FUNCTION_BLOCK PUBLIC FB_Recipe
VAR_INPUT
	bCreateRecipe		: BOOL;
	bEditRecipe         : BOOL;
	bDeleteRecipe		: BOOL;
	tHeatSetTime		: TIME;
	tQuenchTime			: TIME;
	sRecipeName			: STRING(20);
	stRecipeIn			: ST_Recipe;
END_VAR

VAR_OUTPUT
	stRecipeOut			: ST_Recipe;
END_VAR

VAR
	nCounter_1			: INT;
	nMaxRecipes			: INT := 100;
END_VAR

VAR PERSISTENT 
    aRecipeBook			: ARRAY[1..100] OF ST_Recipe;
	aRecipeNames		: ARRAY[1..100] OF STRING(20);
END_VAR

METHOD M_Create : ST_Recipe
VAR_INPUT
	sName				: STRING(20);
	tIngredient_1 		: TIME;
	tIngredient_2 		: TIME;
	
END_VAR
VAR_OUTPUT
	bCreateSuceessful	:BOOL;
	sErrorMsg			:STRING(30) := 'None';
END_VAR
VAR
	stRecipe			: ST_Recipe;
	nCounter			: INT;
	bDuplicateFound		: BOOL;
END_VAR
// check for duplicates
WHILE NOT (bDuplicateFound) AND (nCounter <= nMaxRecipes) DO
	FOR nCounter := 1 TO nMaxRecipes DO
		IF aRecipeBook[nCounter].sRecipeName = sName THEN
			bDuplicateFound := TRUE;
			sErrorMsg := 'Duplicate recipe name found';
			bCreateSuceessful := FALSE;
		END_IF
	END_FOR
END_WHILE

// check recipe array for empty spot
IF NOT bDuplicateFound THEN
	nCounter := 1;
	WHILE (aRecipeBook[nCounter].sRecipeName <> '') AND (nCounter <= nMaxRecipes) DO
		nCounter := nCounter + 1;
	END_WHILE
	
	// check for full recipe array
	IF nCounter > nMaxRecipes THEN
		sErrorMsg := 'Recipe book full';
		bCreateSuceessful := FALSE;
		
	// if no duplicates, fill next available recipe slot	
	ELSIF NOT bDuplicateFound THEN
		stRecipe.sRecipeName := sName;
		stRecipe.tHeatSetTime := tIngredient_1;
		stRecipe.tQuenchTime := tIngredient_2;
		aRecipeBook[nCounter] := stRecipe;
		bCreateSuceessful := TRUE;
		M_UpdateRecipeNames();
	END_IF
END_IF
END_METHOD

METHOD M_Delete : BOOL
VAR_INPUT
	sName				: STRING(20);
END_VAR
VAR_OUTPUT
	bDeleteSuccessful 	: BOOL;
END_VAR
VAR
	nCounter 			: INT;
END_VAR
nCounter := 1;
WHILE (aRecipeBook[nCounter].sRecipeName <> sName) AND (nCounter <= nMaxRecipes) DO
	nCounter := nCounter + 1;
END_WHILE

IF nCounter > nMaxRecipes THEN
	bDeleteSuccessful := FALSE;
ELSE
	aRecipeBook[nCounter].sRecipeName := '';
	aRecipeBook[nCounter].tHeatSetTime := T#0S;
	aRecipeBook[nCounter].tQuenchTime := T#0S;
	bDeleteSuccessful := TRUE;
	M_UpdateRecipeNames();
END_IF
END_METHOD

METHOD M_Edit : BOOL
VAR_INPUT
	sName				: STRING(20);
	tNewIngredient_1 	: TIME;
	tNewIngredient_2 	: TIME;
END_VAR
VAR_OUTPUT
	bEditSuccessful 	: BOOL;
	sErrorMsg			: STRING(30);
	stRecipeOut			: ST_Recipe;
END_VAR
VAR
	nCounter			: INT := 1;
END_VAR
// find recipe in recipe book
WHILE (aRecipeBook[nCounter].sRecipeName <> sName) AND (nCounter <= nMaxRecipes) DO
	nCounter := nCounter + 1;
END_WHILE

// check if recipe not found
IF nCounter > nMaxRecipes THEN
	sErrorMsg := 'Recipe not found';
	bEditSuccessful := FALSE;
	
// update time values
ELSE
	aRecipeBook[nCounter].tHeatSetTime := tNewIngredient_1;
	aRecipeBook[nCounter].tQuenchTime := tNewIngredient_2;
END_IF
END_METHOD

METHOD M_OrderList : BOOL
VAR_INPUT
	sName			: STRING(20);
END_VAR
VAR
	nCounter		: INT := 1;
	nStrLen_1		: INT;
	nStrLen_2		: INT;
	sString_1		: STRING(20);
	sString_2		: STRING(20);
	sPlaceholder	: STRING(20);
END_VAR
WHILE nCounter < nMaxRecipes DO
	// store nth and nth + 1 string as uppercase
	sString_1 := aRecipeNames[nCounter];
	sString_2 := aRecipeNames[nCounter + 1];
	sString_1 := F_ToUCase(sString_1);
	sString_2 := F_ToUCase(sString_2);
	
	// store string lengths
	nStrLen_1 := LEN(STR := sString_1);
	nStrLen_2 := LEN(STR := sString_2);
	
	// check if 1st string empty and 2nd string not
	IF nStrLen_1 = 0 AND nStrLen_2 <> 0 THEN
		// replcae 1st str with 2nd str
		aRecipeNames[nCounter] := sString_2;
	
	// check if both values are 0
	ELSIF nStrLen_1 = 0 AND nStrLen_2 = 0 THEN
		EXIT;
		
	// check if 1st string 1st char is less than 2nd string 1st char
	ELSIF LEFT(STR := sString_1, SIZE := 1) < LEFT(STR := sString_2, SIZE := 1) THEN 
		// swap names
		sPlaceholder := sString_1;
		aRecipeNames[nCounter] := sString_2;
		aRecipeNames[nCounter + 1] := sPlaceholder;
		nCounter := 1;
	END_IF
	nCounter := nCounter + 1;
END_WHILE
END_METHOD

METHOD M_UpdateRecipeNames : BOOL
VAR_INPUT
END_VAR
VAR
	nItem	: INT;
	nIndex	: INT := 1;
END_VAR
FOR nItem := 1 TO nMaxRecipes DO
	IF aRecipeBook[nItem].sRecipeName <> '' THEN
		aRecipeNames[nIndex] := aRecipeBook[nItem].sRecipeName;
		nIndex := nIndex + 1;
	END_IF
END_FOR
END_METHOD

END_FUNCTION_BLOCK

(* stored: Version 1.1.0.1, ProductVersion 3.1.4024.11
   POU FB_Recipe: Id {b4198a36-65da-4222-8d3e-14fa98442687}, SpecialFunc None
   Method M_Create: Id {789aa0a5-f168-4631-a4e5-4b7480ae637c}
   Method M_Delete: Id {9a285bd6-1b35-4cdf-8070-246e1f8a2082}
   Method M_Edit: Id {36cee79e-3e26-448d-a779-b9438a128454}
   Method M_OrderList: Id {392bedb9-e486-4e01-b047-423d7d7c7ecc}
   Method M_UpdateRecipeNames: Id {159f407e-1f95-465b-a3f5-231de04b49d7} *)
